// TIA Portal V17 export
// export: Created 2023-12-22T15:05:26.6725301Z, ExportSetting WithDefaults, DisplayName Totally Integrated Automation Portal, DisplayVersion V17, DisplayName TIA Portal Openness, DisplayVersion V17, DisplayName TIA Portal Version Control Interface, DisplayVersion V17, DisplayName STEP 7 Professional, DisplayVersion V17, DisplayName STEP 7 Safety, DisplayVersion V17, DisplayName WinCC Advanced, DisplayVersion V17
FUNCTION_BLOCK "AO_ex"   // FB104, LAD
{ S7_Optimized_Access := 'FALSE' }
VERSION : 0.1
// stored: AutoNumber false, IsIECCheckEnabled false, SetENOAutomatically false, UDAEnableTagReadback false
   VAR_INPUT
      SP_A : Real;   // Уставка авторежима
      All_Block : Bool;   // Аварийная остановка
   END_VAR
   VAR_IN_OUT
      Signal : Int;   // Входной сигнал контроллера
   END_VAR
   VAR DB_SPECIFIC
      CMD : "CMD";   // Основные команды / Блок команд
      Mode : Int;   // Режим работы
      Status : Int;   // Статус устройства
      Use : Struct   // Функционал
         Indirect { S7_SetPoint := 'True'} : Bool := true;   // Косвенная адресация
      END_STRUCT;
      VmA : Real;   // Реальный сигнал на входе ПЛК
      SP_M : Real;   // Уставка в ручном режиме
   END_VAR
   VAR
      Converter { S7_SetPoint := 'True'} : "Converter";   // Масштабирование сигнала
   END_VAR
   VAR DB_SPECIFIC
      Events : Word;   // События датчика
      pos : Array[0..15] of Bool;   // Контроль фронтов событий
      Output_Type { S7_SetPoint := 'True'} : Int;   // Тип выхода, 0 - 4..20, 1 - 0..20, 2 - 0..10, 3 - 0..5
      CodeID { S7_SetPoint := 'True'} : Int;   // Код датчика для привязки в скаде
      "Type" { S7_SetPoint := 'True'} : Int;   // Тип датчика (единицы измерения)
      ADDR { S7_SetPoint := 'True'} : Int;   // Адрес выхода на контроллере
   END_VAR
   VAR
      Slow { S7_SetPoint := 'True'} : "Slow";   // Плавное управление
   END_VAR
   VAR DB_SPECIFIC
      Time_DTL { S7_SetPoint := 'True'} : DTL;
   END_VAR
   VAR_TEMP
      ev : Bool;   // флаг управления событиями
      Signal_R : Real;   // Актуальный сигнал
      Signal_Ex : Real;   // Конвертация сигнала
      Signal_Dint : DInt;   // Сигнал в DInt
      Type_Min : Real;
      Type_Max : Real;
   END_VAR
   // CMD.Start_A := true;
   VAR_TEMP   // added for the SCL form of the ladder/FBD networks
      _w1 : Bool;
      _w2 : Bool;
      _w3 : Bool;
      _w4 : Bool;
      _w5 : Bool;
      _w6 : Bool;
      _w7 : Bool;
      _w8 : Bool;
      _w9 : Bool;
      _w10 : Bool;
      _w11 : Bool;
      _w12 : Bool;
      _w13 : Bool;
      _w14 : Bool;
      _w15 : Bool;
      _w16 : Bool;
   END_VAR
BEGIN

REGION Network 1: Устройство в ручном режиме
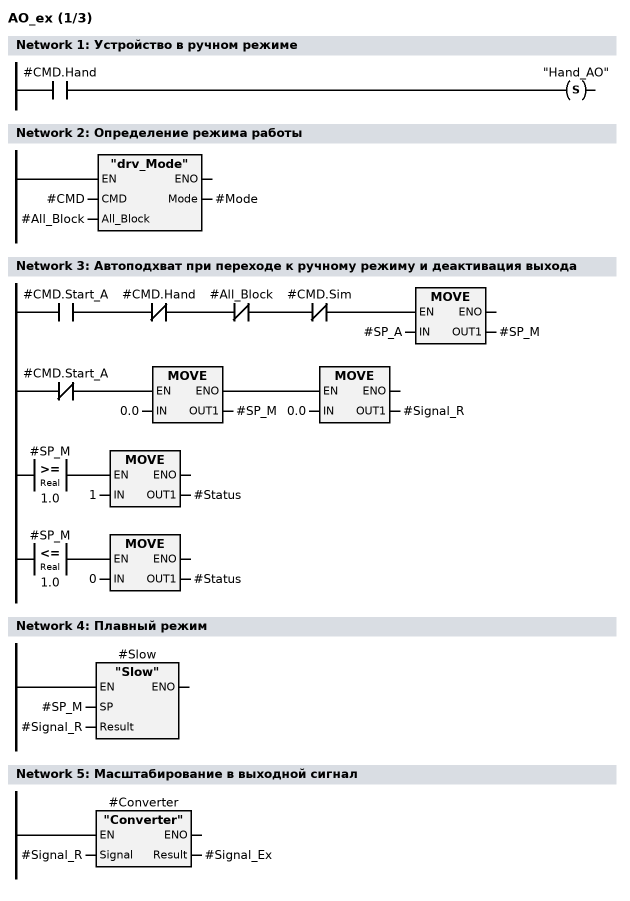
   RUNG wire#powerrail
      Contact( #CMD.Hand )
      S_Coil( "Hand_AO" )
   END_RUNG
   // the same network as SCL:
   IF #CMD.Hand THEN "Hand_AO" := TRUE; END_IF;
END_REGION

REGION Network 2: Определение режима работы
   RUNG wire#powerrail
      "drv_Mode"(CMD := #CMD, All_Block := #All_Block, Mode => #Mode)
   END_RUNG
   // the same network as SCL:
   "drv_Mode"(CMD := #CMD, All_Block := #All_Block, Mode => #Mode);
END_REGION

REGION Network 3: Автоподхват при переходе к ручному режиму и деактивация выхода
   RUNG wire#powerrail
      Contact( #CMD.Start_A )
      I_Contact( #CMD.Hand )
      I_Contact( #All_Block )
      I_Contact( #CMD.Sim )
      { S7_GenerateENO := "TRUE" } Move(in := #SP_A, out1 => #SP_M)
   END_RUNG
   RUNG wire#powerrail
      I_Contact( #CMD.Start_A )
      { S7_GenerateENO := "TRUE" } Move(in := 0.0, out1 => #SP_M)
      { S7_GenerateENO := "TRUE" } Move(in := 0.0, out1 => #Signal_R)
   END_RUNG
   RUNG wire#powerrail
      { S7_Templates := "SrcType := Real" } GE_Contact(in1 := #SP_M, in2 := 1.0)
      Move(in := 1, out1 => #Status)
   END_RUNG
   RUNG wire#powerrail
      { S7_Templates := "SrcType := Real" } LE_Contact(in1 := #SP_M, in2 := 1.0)
      Move(in := 0, out1 => #Status)
   END_RUNG
   // the same network as SCL:
   // ENO of a box is taken as its EN; it also drops when the box reports an error
   IF #CMD.Start_A AND NOT #CMD.Hand AND NOT #All_Block AND NOT #CMD.Sim THEN #SP_M := #SP_A; END_IF;
   IF NOT #CMD.Start_A THEN
       #SP_M := 0.0;
       #Signal_R := 0.0;
   END_IF;
   IF #SP_M >= 1.0 THEN #Status := 1; END_IF;
   IF #SP_M <= 1.0 THEN #Status := 0; END_IF;
END_REGION

REGION Network 4: Плавный режим
   RUNG wire#powerrail
      #Slow(SP := #SP_M, Result := #Signal_R)
   END_RUNG
   // the same network as SCL:
   #Slow(SP := #SP_M, Result := #Signal_R);   // "Slow"
END_REGION

REGION Network 5: Масштабирование в выходной сигнал
   RUNG wire#powerrail
      #Converter(Signal := #Signal_R, Result => #Signal_Ex)
   END_RUNG
   // the same network as SCL:
   #Converter(Signal := #Signal_R, Result => #Signal_Ex);   // "Converter"
END_REGION

REGION Network 6: Преобразование кода в реальное значение входа
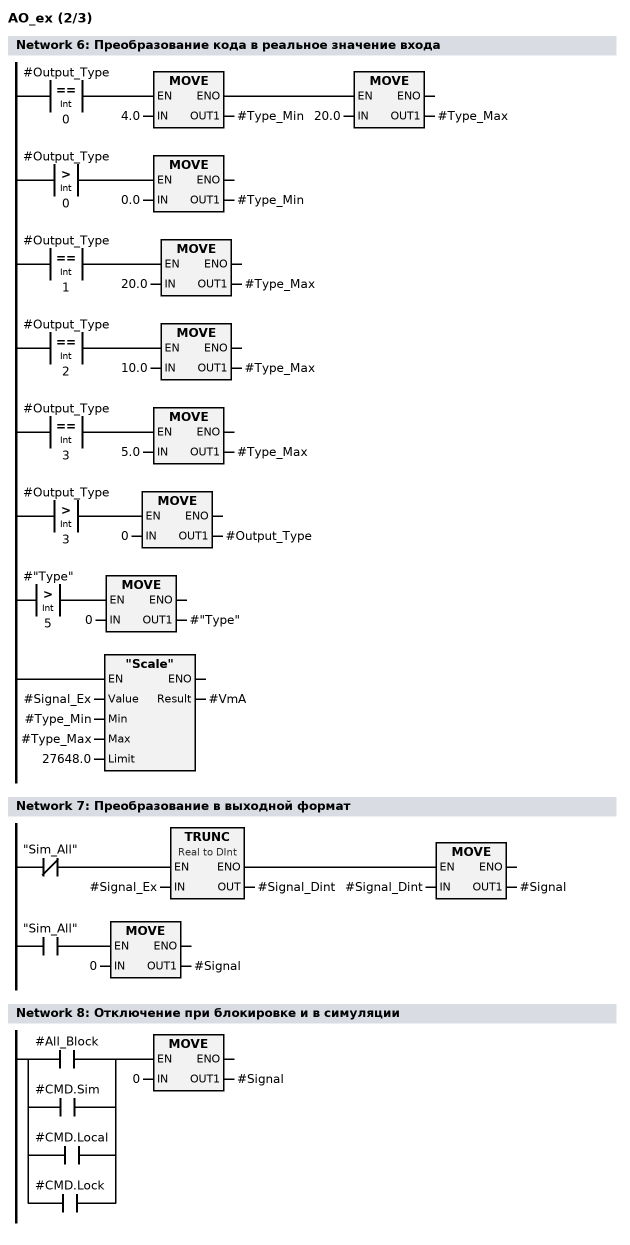
   RUNG wire#powerrail
      { S7_Templates := "SrcType := Int" } EQ_Contact(in1 := #Output_Type, in2 := 0)
      Move(in := 4.0, out1 => #Type_Min)
      Move(in := 20.0, out1 => #Type_Max)
   END_RUNG
   RUNG wire#powerrail
      { S7_Templates := "SrcType := Int" } GT_Contact(in1 := #Output_Type, in2 := 0)
      Move(in := 0.0, out1 => #Type_Min)
   END_RUNG
   RUNG wire#powerrail
      { S7_Templates := "SrcType := Int" } EQ_Contact(in1 := #Output_Type, in2 := 1)
      Move(in := 20.0, out1 => #Type_Max)
   END_RUNG
   RUNG wire#powerrail
      { S7_Templates := "SrcType := Int" } EQ_Contact(in1 := #Output_Type, in2 := 2)
      Move(in := 10.0, out1 => #Type_Max)
   END_RUNG
   RUNG wire#powerrail
      { S7_Templates := "SrcType := Int" } EQ_Contact(in1 := #Output_Type, in2 := 3)
      Move(in := 5.0, out1 => #Type_Max)
   END_RUNG
   RUNG wire#powerrail
      { S7_Templates := "SrcType := Int" } GT_Contact(in1 := #Output_Type, in2 := 3)
      Move(in := 0, out1 => #Output_Type)
   END_RUNG
   RUNG wire#powerrail
      { S7_Templates := "SrcType := Int" } GT_Contact(in1 := #"Type", in2 := 5)
      Move(in := 0, out1 => #"Type")
   END_RUNG
   RUNG wire#powerrail
      "Scale"(Value := #Signal_Ex, Min := #Type_Min, Max := #Type_Max, Limit := 27648.0, Result => #VmA)
   END_RUNG
   // the same network as SCL:
   IF #Output_Type = 0 THEN
       #Type_Min := 4.0;
       #Type_Max := 20.0;
   END_IF;
   IF #Output_Type > 0 THEN #Type_Min := 0.0; END_IF;
   IF #Output_Type = 1 THEN #Type_Max := 20.0; END_IF;
   IF #Output_Type = 2 THEN #Type_Max := 10.0; END_IF;
   IF #Output_Type = 3 THEN #Type_Max := 5.0; END_IF;
   IF #Output_Type > 3 THEN #Output_Type := 0; END_IF;
   IF #"Type" > 5 THEN #"Type" := 0; END_IF;
   "Scale"(Value := #Signal_Ex, Min := #Type_Min, Max := #Type_Max, Limit := 27648.0, Result => #VmA);
END_REGION

REGION Network 7: Преобразование в выходной формат
   RUNG wire#powerrail
      I_Contact( "Sim_All" )
      { S7_Templates := "[SrcType := Real, DestType := DInt]"; S7_GenerateENO := "TRUE" } Trunc(in := #Signal_Ex, out => #Signal_Dint)
      { S7_GenerateENO := "TRUE" } Move(in := #Signal_Dint, out1 => #Signal)
   END_RUNG
   RUNG wire#powerrail
      Contact( "Sim_All" )
      { S7_GenerateENO := "TRUE" } Move(in := 0, out1 => #Signal)
   END_RUNG
   // the same network as SCL:
   // ENO of a box is taken as its EN; it also drops when the box reports an error
   IF NOT "Sim_All" THEN
       #Signal_Dint := TRUNC(#Signal_Ex);
       #Signal := #Signal_Dint;
   END_IF;
   IF "Sim_All" THEN #Signal := 0; END_IF;
END_REGION

REGION Network 8: Отключение при блокировке и в симуляции
   RUNG wire#powerrail
      Contact( #All_Block )
      wire#w1
      { S7_GenerateENO := "TRUE" } Move(in := 0, out1 => #Signal)
   END_RUNG
   RUNG wire#powerrail
      Contact( #CMD.Sim )
   END_RUNG wire#w1
   RUNG wire#powerrail
      Contact( #CMD.Local )
   END_RUNG wire#w1
   RUNG wire#powerrail
      Contact( #CMD.Lock )
   END_RUNG wire#w1
   // the same network as SCL:
   IF #All_Block OR #CMD.Sim OR #CMD.Local OR #CMD.Lock THEN #Signal := 0; END_IF;
END_REGION

REGION Network 9: События выхода
   // 0 - выход активирован
   // 1 - выход деактивирован
   // 2 - выход в ручном режиме
   // 3 - выход в автоматическом режиме
   // 4 - плавный разгон активирован
   // 5 - плавный разгон деактивирован
   // 6 - плавное замедление активировано
   // 7 - плавное замедление деактивировано
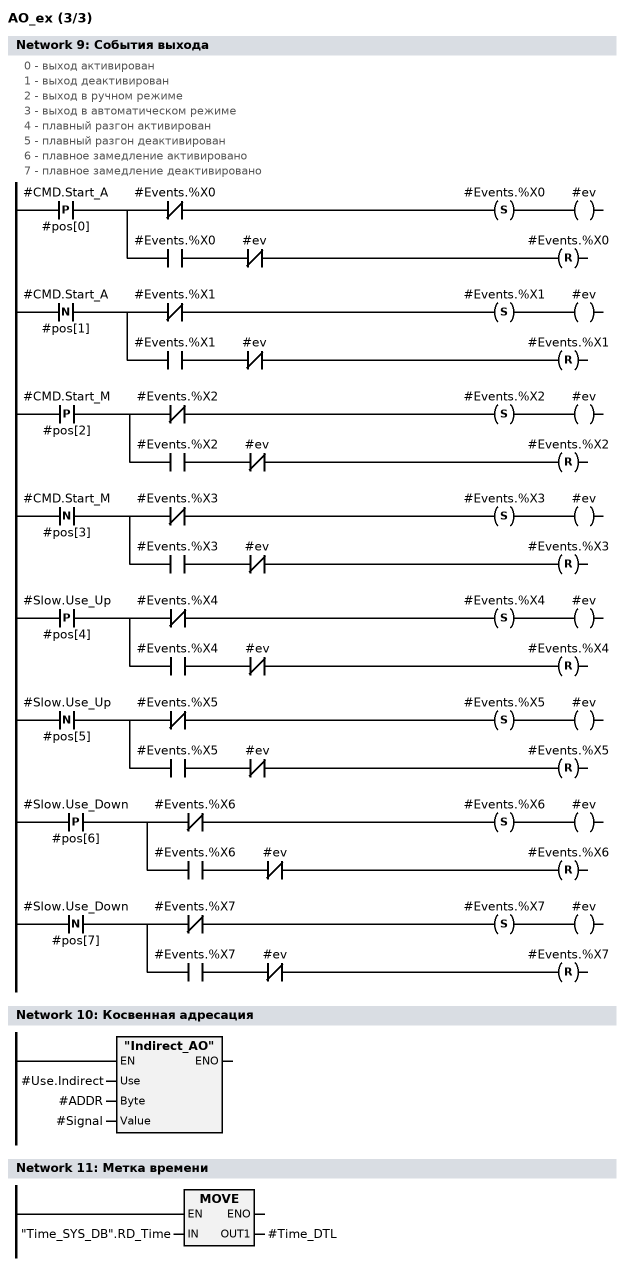
   RUNG wire#powerrail
      P_Contact(operand := #CMD.Start_A, bit := #pos[0])
      wire#w1
      I_Contact( #Events.%X0 )
      S_Coil( #Events.%X0 )
      Coil( #ev )
   END_RUNG
   RUNG wire#w1
      Contact( #Events.%X0 )
      I_Contact( #ev )
      R_Coil( #Events.%X0 )
   END_RUNG
   RUNG wire#powerrail
      N_Contact(operand := #CMD.Start_A, bit := #pos[1])
      wire#w2
      I_Contact( #Events.%X1 )
      S_Coil( #Events.%X1 )
      Coil( #ev )
   END_RUNG
   RUNG wire#w2
      Contact( #Events.%X1 )
      I_Contact( #ev )
      R_Coil( #Events.%X1 )
   END_RUNG
   RUNG wire#powerrail
      P_Contact(operand := #CMD.Start_M, bit := #pos[2])
      wire#w3
      I_Contact( #Events.%X2 )
      S_Coil( #Events.%X2 )
      Coil( #ev )
   END_RUNG
   RUNG wire#w3
      Contact( #Events.%X2 )
      I_Contact( #ev )
      R_Coil( #Events.%X2 )
   END_RUNG
   RUNG wire#powerrail
      N_Contact(operand := #CMD.Start_M, bit := #pos[3])
      wire#w4
      I_Contact( #Events.%X3 )
      S_Coil( #Events.%X3 )
      Coil( #ev )
   END_RUNG
   RUNG wire#w4
      Contact( #Events.%X3 )
      I_Contact( #ev )
      R_Coil( #Events.%X3 )
   END_RUNG
   RUNG wire#powerrail
      P_Contact(operand := #Slow.Use_Up, bit := #pos[4])
      wire#w5
      I_Contact( #Events.%X4 )
      S_Coil( #Events.%X4 )
      Coil( #ev )
   END_RUNG
   RUNG wire#w5
      Contact( #Events.%X4 )
      I_Contact( #ev )
      R_Coil( #Events.%X4 )
   END_RUNG
   RUNG wire#powerrail
      N_Contact(operand := #Slow.Use_Up, bit := #pos[5])
      wire#w6
      I_Contact( #Events.%X5 )
      S_Coil( #Events.%X5 )
      Coil( #ev )
   END_RUNG
   RUNG wire#w6
      Contact( #Events.%X5 )
      I_Contact( #ev )
      R_Coil( #Events.%X5 )
   END_RUNG
   RUNG wire#powerrail
      P_Contact(operand := #Slow.Use_Down, bit := #pos[6])
      wire#w7
      I_Contact( #Events.%X6 )
      S_Coil( #Events.%X6 )
      Coil( #ev )
   END_RUNG
   RUNG wire#w7
      Contact( #Events.%X6 )
      I_Contact( #ev )
      R_Coil( #Events.%X6 )
   END_RUNG
   RUNG wire#powerrail
      N_Contact(operand := #Slow.Use_Down, bit := #pos[7])
      wire#w8
      I_Contact( #Events.%X7 )
      S_Coil( #Events.%X7 )
      Coil( #ev )
   END_RUNG
   RUNG wire#w8
      Contact( #Events.%X7 )
      I_Contact( #ev )
      R_Coil( #Events.%X7 )
   END_RUNG
   // the same network as SCL:
   #_w1 := #CMD.Start_A AND NOT #pos[0];   // rising edge of #CMD.Start_A
   #pos[0] := #CMD.Start_A;
   #_w2 := #_w1 AND NOT #Events.%X0;
   IF #_w2 THEN #Events.%X0 := TRUE; END_IF;
   #ev := #_w2;
   IF #_w1 AND #Events.%X0 AND NOT #ev THEN #Events.%X0 := FALSE; END_IF;
   #_w3 := NOT #CMD.Start_A AND #pos[1];   // falling edge of #CMD.Start_A
   #pos[1] := #CMD.Start_A;
   #_w4 := #_w3 AND NOT #Events.%X1;
   IF #_w4 THEN #Events.%X1 := TRUE; END_IF;
   #ev := #_w4;
   IF #_w3 AND #Events.%X1 AND NOT #ev THEN #Events.%X1 := FALSE; END_IF;
   #_w5 := #CMD.Start_M AND NOT #pos[2];   // rising edge of #CMD.Start_M
   #pos[2] := #CMD.Start_M;
   #_w6 := #_w5 AND NOT #Events.%X2;
   IF #_w6 THEN #Events.%X2 := TRUE; END_IF;
   #ev := #_w6;
   IF #_w5 AND #Events.%X2 AND NOT #ev THEN #Events.%X2 := FALSE; END_IF;
   #_w7 := NOT #CMD.Start_M AND #pos[3];   // falling edge of #CMD.Start_M
   #pos[3] := #CMD.Start_M;
   #_w8 := #_w7 AND NOT #Events.%X3;
   IF #_w8 THEN #Events.%X3 := TRUE; END_IF;
   #ev := #_w8;
   IF #_w7 AND #Events.%X3 AND NOT #ev THEN #Events.%X3 := FALSE; END_IF;
   #_w9 := #Slow.Use_Up AND NOT #pos[4];   // rising edge of #Slow.Use_Up
   #pos[4] := #Slow.Use_Up;
   #_w10 := #_w9 AND NOT #Events.%X4;
   IF #_w10 THEN #Events.%X4 := TRUE; END_IF;
   #ev := #_w10;
   IF #_w9 AND #Events.%X4 AND NOT #ev THEN #Events.%X4 := FALSE; END_IF;
   #_w11 := NOT #Slow.Use_Up AND #pos[5];   // falling edge of #Slow.Use_Up
   #pos[5] := #Slow.Use_Up;
   #_w12 := #_w11 AND NOT #Events.%X5;
   IF #_w12 THEN #Events.%X5 := TRUE; END_IF;
   #ev := #_w12;
   IF #_w11 AND #Events.%X5 AND NOT #ev THEN #Events.%X5 := FALSE; END_IF;
   #_w13 := #Slow.Use_Down AND NOT #pos[6];   // rising edge of #Slow.Use_Down
   #pos[6] := #Slow.Use_Down;
   #_w14 := #_w13 AND NOT #Events.%X6;
   IF #_w14 THEN #Events.%X6 := TRUE; END_IF;
   #ev := #_w14;
   IF #_w13 AND #Events.%X6 AND NOT #ev THEN #Events.%X6 := FALSE; END_IF;
   #_w15 := NOT #Slow.Use_Down AND #pos[7];   // falling edge of #Slow.Use_Down
   #pos[7] := #Slow.Use_Down;
   #_w16 := #_w15 AND NOT #Events.%X7;
   IF #_w16 THEN #Events.%X7 := TRUE; END_IF;
   #ev := #_w16;
   IF #_w15 AND #Events.%X7 AND NOT #ev THEN #Events.%X7 := FALSE; END_IF;
END_REGION

REGION Network 10: Косвенная адресация
   RUNG wire#powerrail
      "Indirect_AO"(Use := #Use.Indirect, "Byte" := #ADDR, Value := #Signal)
   END_RUNG
   // the same network as SCL:
   "Indirect_AO"(Use := #Use.Indirect, "Byte" := #ADDR, Value := #Signal);
END_REGION

REGION Network 11: Метка времени
   RUNG wire#powerrail
      Move(in := "Time_SYS_DB".RD_Time, out1 => #Time_DTL)
   END_RUNG
   // the same network as SCL:
   #Time_DTL := "Time_SYS_DB".RD_Time;
END_REGION
END_FUNCTION_BLOCK
